(* LS Electric XG5000 project: test1 *)
(* PLC LSPLC *)
(* module base 0 slot 0: 입출력 모듈:XGH-DT4A (DC 24V 입력, 트랜지스터 출력 32점 ) *)

PROGRAM NewProgram (* task: 스캔 프로그램 *)
VAR
    리셋 : BOOL;
    모터1 : BOOL;
    모터2 : BOOL;
    모터3 : BOOL;
    셧아웃 : BOOL;
    셧아웃2 : BOOL;
    셧아웃3 : BOOL;
    스위치1 : BOOL;
END_VAR
VAR
    _e1 : R_TRIG;
    _e2 : R_TRIG;
    _e3 : R_TRIG;
    _e4 : R_TRIG;
    _e5 : R_TRIG;
    _e6 : R_TRIG;
    _e7 : R_TRIG;
    _p8 : BOOL;
    _e9 : R_TRIG;
    _e10 : R_TRIG;
    _e11 : R_TRIG;
    _e12 : R_TRIG;
    _p13 : BOOL;
    _e14 : R_TRIG;
    _e15 : R_TRIG;
    _e16 : R_TRIG;
    _e17 : R_TRIG;
    _p18 : BOOL;
    _e19 : R_TRIG;
END_VAR

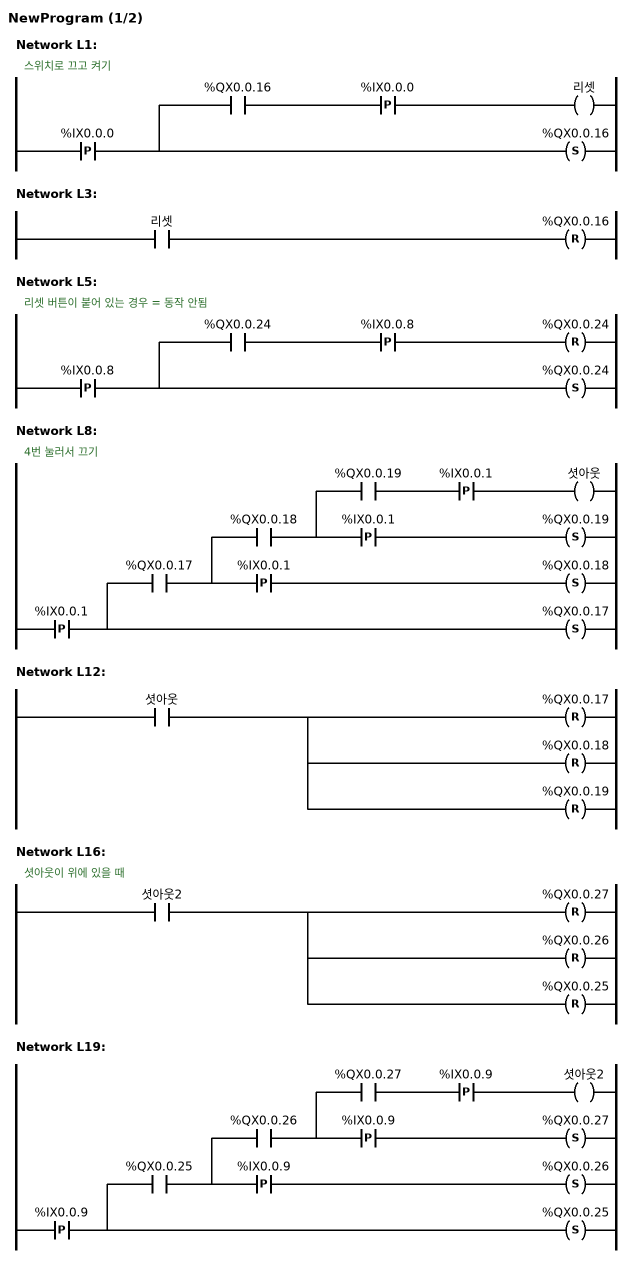
(* 스위치로 끄고 켜기 *)
(* Rung L1 *)
_e1(CLK := %IX0.0.0);
_e2(CLK := %IX0.0.0);
리셋 := _e1.Q AND %QX0.0.16 AND _e2.Q;
IF _e1.Q THEN %QX0.0.16 := TRUE; END_IF;
(* Rung L3 *)
IF 리셋 THEN %QX0.0.16 := FALSE; END_IF;
(* 리셋 버튼이 붙어 있는 경우 = 동작 안됨 *)
(* Rung L5 *)
_e3(CLK := %IX0.0.8);
_e4(CLK := %IX0.0.8);
IF _e3.Q AND %QX0.0.24 AND _e4.Q THEN %QX0.0.24 := FALSE; END_IF;
IF _e3.Q THEN %QX0.0.24 := TRUE; END_IF;
(* 4번 눌러서 끄기 *)
(* Rung L8 *)
_e5(CLK := %IX0.0.1);
_e6(CLK := %IX0.0.1);
셧아웃 := _e5.Q AND %QX0.0.17 AND %QX0.0.18 AND %QX0.0.19 AND _e6.Q;
_e7(CLK := %IX0.0.1);
_p8 := _e5.Q AND %QX0.0.17;
IF _e5.Q AND %QX0.0.17 AND %QX0.0.18 AND _e7.Q THEN %QX0.0.19 := TRUE; END_IF;
_e9(CLK := %IX0.0.1);
IF _p8 AND _e9.Q THEN %QX0.0.18 := TRUE; END_IF;
IF _e5.Q THEN %QX0.0.17 := TRUE; END_IF;
(* Rung L12 *)
IF 셧아웃 THEN
    %QX0.0.17 := FALSE;
    %QX0.0.18 := FALSE;
    %QX0.0.19 := FALSE;
END_IF;
(* 셧아웃이 위에 있을 때 *)
(* Rung L16 *)
IF 셧아웃2 THEN
    %QX0.0.27 := FALSE;
    %QX0.0.26 := FALSE;
    %QX0.0.25 := FALSE;
END_IF;
(* Rung L19 *)
_e10(CLK := %IX0.0.9);
_e11(CLK := %IX0.0.9);
셧아웃2 := _e10.Q AND %QX0.0.25 AND %QX0.0.26 AND %QX0.0.27 AND _e11.Q;
_e12(CLK := %IX0.0.9);
_p13 := _e10.Q AND %QX0.0.25;
IF _e10.Q AND %QX0.0.25 AND %QX0.0.26 AND _e12.Q THEN %QX0.0.27 := TRUE; END_IF;
_e14(CLK := %IX0.0.9);
IF _p13 AND _e14.Q THEN %QX0.0.26 := TRUE; END_IF;
IF _e10.Q THEN %QX0.0.25 := TRUE; END_IF;

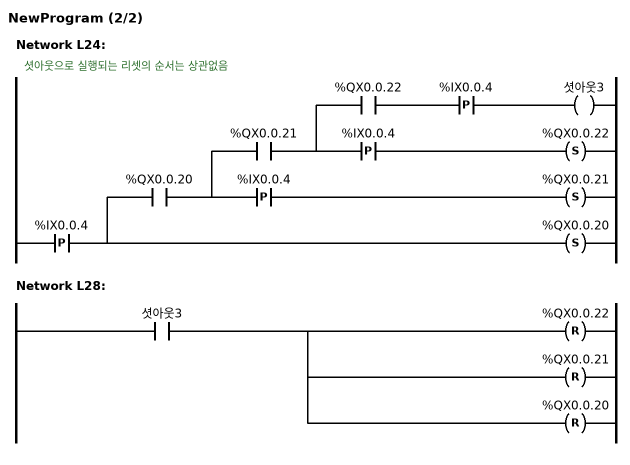
(* 셧아웃으로 실행되는 리셋의 순서는 상관없음 *)
(* Rung L24 *)
_e15(CLK := %IX0.0.4);
_e16(CLK := %IX0.0.4);
셧아웃3 := _e15.Q AND %QX0.0.20 AND %QX0.0.21 AND %QX0.0.22 AND _e16.Q;
_e17(CLK := %IX0.0.4);
_p18 := _e15.Q AND %QX0.0.20;
IF _e15.Q AND %QX0.0.20 AND %QX0.0.21 AND _e17.Q THEN %QX0.0.22 := TRUE; END_IF;
_e19(CLK := %IX0.0.4);
IF _p18 AND _e19.Q THEN %QX0.0.21 := TRUE; END_IF;
IF _e15.Q THEN %QX0.0.20 := TRUE; END_IF;
(* Rung L28 *)
IF 셧아웃3 THEN
    %QX0.0.22 := FALSE;
    %QX0.0.21 := FALSE;
    %QX0.0.20 := FALSE;
END_IF;
END_PROGRAM